# EPICS substitutions: iocs/aerotechIOC/iocBoot/iocAerotech/Soloist.substitutions
file "$(MOTOR)/db/motor.db"
{
pattern
{P,             N,       M,        DTYP,        C,      S,      DESC,           EGU,            DIR,    VELO,   VBAS,   ACCL,   BDST,   BVEL,   BACC,   MRES,   PREC,   DHLM,   DLLM,   INIT}
{aerotech:,     2,     "m$(N)",  "Soloist",     0,      0,      "motor $(N)",   degrees,        Pos,    1,      .1,     .2,     0,      1,       .2,    2.5e-4, 5,      100,    -100,   ""}
}
